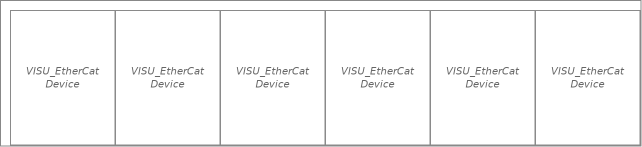
VISUALIZATION VISU_HydraulicsPumpsGroupIO  // 642x147
VAR_IN_OUT
	ref : HydraulicsPumpsGroupIO;
    widget : HydraulicsPumpsGroupIOWidget;
END_VAR
    Frame (10,10 105x135)
        shows VISU_EtherCatDevice(device := ref.parts.COU, widget := widget.COU)
    Frame (115,10 105x135)
        shows VISU_EtherCatDevice(device := ref.parts.DI1, widget := widget.DI1)
    Frame (220,10 105x135)
        shows VISU_EtherCatDevice(device := ref.parts.SI1, widget := widget.SI1)
    Frame (325,10 105x135)
        shows VISU_EtherCatDevice(device := ref.parts.SI2, widget := widget.SI2)
    Frame (430,10 105x135)
        shows VISU_EtherCatDevice(device := ref.parts.SI3, widget := widget.SI3)
    Frame (535,10 105x135)
        shows VISU_EtherCatDevice(device := ref.parts.DI2, widget := widget.DI2)
END_VISUALIZATION

(* stored: Version 1.1.0.1, ProductVersion 3.1.4019.2
   Visu VISU_HydraulicsPumpsGroupIO: Id {4bef8f03-ec29-477c-a6a7-6eaa0b81cf14} *)
